{attribute 'GeneratedUsingTerminal: IODEVICETYPE_ETHERCATPROT'}
{attribute addProperty BoxType "IODEVICETYPE_ETHERCATPROT"}
{attribute addProperty Id "Beckhoff_EL1xxxBeckhoff_EL1xxx_3E37AACA6236Beckhoff_EL2xxxBeckhoff_EL2xxx_F4C539CA2992Beckhoff_EL3xxxBeckhoff_EL3xxx_05984D3D1813Beckhoff_EL3xxx_0030Beckhoff_EL3xxx_0030_EF742EC0265Beckhoff_EL4xxxBeckhoff_EL4xxx_BC7C1D702405Beckhoff_EL5xxxBeckhoff_EL5xxx_A510F2723086Beckhoff_EL6xxxBeckhoff_EL6xxx_5832F4A84115Beckhoff_EL7xxxBeckhoff_EL7xxx_96878FD52666Beckhoff_EL9xxxBeckhoff_EL9xxx_9771C92C1254Beckhoff_EL15xxBeckhoff_EL15xx_7FFDF3B3529Beckhoff_EL19xxBeckhoff_EL19xx_C9550BF750Beckhoff_EL25xxBeckhoff_EL25xx_A1E3F9182720Beckhoff_EL29xxBeckhoff_EL29xx_FCC67B4476Beckhoff_EL30xxBeckhoff_EL30xx_D5E79B105129Beckhoff_EL31xxBeckhoff_EL31xx_098DC56E3694Beckhoff_EL32xxBeckhoff_EL32xx_152143682581Beckhoff_EL33xxBeckhoff_EL33xx_7753F1402459Beckhoff_EL34xxBeckhoff_EL34xx_5C8507D711825Beckhoff_EL37xxBeckhoff_EL37xx_E7914E0E2253Beckhoff_EL47xxBeckhoff_EL47xx_F9F61196294Beckhoff_EL66xxBeckhoff_EL66xx_32F43B791034Beckhoff_EL67xxBeckhoff_EL67xx_9D033AAA966Beckhoff_EL68xxBeckhoff_EL68xx_6F2062753597Beckhoff_EL69xxBeckhoff_EL69xx_55DE5C9C198Beckhoff_EL72xxBeckhoff_EL72xx_566ED46D3383Beckhoff_EL73xxBeckhoff_EL73xx_3D4E24E01278Beckhoff_EL99xxBeckhoff_EL99xx_FA66A12D10SyncUnitsSyncUnits_9F8710E11242InputsInputs_25A0042B160OutputsOutputs_2397A10E106InfoDataInfoData_E68C61CD28"}
{attribute addProperty CRC "1261115388"}
{attribute addProperty Size "68444"}
TYPE EtherCAT_Master_ELxxxx_4B2B17FC :
STRUCT
	{attribute addProperty Name "Beckhoff_EL1xxx"}
	Beckhoff_EL1xxx : Beckhoff_EL1xxx_3E37AACA;
	{attribute addProperty Name "Beckhoff_EL2xxx"}
	Beckhoff_EL2xxx : Beckhoff_EL2xxx_F4C539CA;
	{attribute addProperty Name "Beckhoff_EL3xxx"}
	Beckhoff_EL3xxx : Beckhoff_EL3xxx_05984D3D;
	{attribute addProperty Name "Beckhoff_EL3xxx_0030"}
	Beckhoff_EL3xxx_0030 : Beckhoff_EL3xxx_0030_EF742EC0;
	{attribute addProperty Name "Beckhoff_EL4xxx"}
	Beckhoff_EL4xxx : Beckhoff_EL4xxx_BC7C1D70;
	{attribute addProperty Name "Beckhoff_EL5xxx"}
	Beckhoff_EL5xxx : Beckhoff_EL5xxx_A510F272;
	{attribute addProperty Name "Beckhoff_EL6xxx"}
	Beckhoff_EL6xxx : Beckhoff_EL6xxx_5832F4A8;
	{attribute addProperty Name "Beckhoff_EL7xxx"}
	Beckhoff_EL7xxx : Beckhoff_EL7xxx_96878FD5;
	{attribute addProperty Name "Beckhoff_EL9xxx"}
	Beckhoff_EL9xxx : Beckhoff_EL9xxx_9771C92C;
	{attribute addProperty Name "Beckhoff_EL15xx"}
	Beckhoff_EL15xx : Beckhoff_EL15xx_7FFDF3B3;
	{attribute addProperty Name "Beckhoff_EL19xx"}
	Beckhoff_EL19xx : Beckhoff_EL19xx_C9550BF7;
	{attribute addProperty Name "Beckhoff_EL25xx"}
	Beckhoff_EL25xx : Beckhoff_EL25xx_A1E3F918;
	{attribute addProperty Name "Beckhoff_EL29xx"}
	Beckhoff_EL29xx : Beckhoff_EL29xx_FCC67B44;
	{attribute addProperty Name "Beckhoff_EL30xx"}
	Beckhoff_EL30xx : Beckhoff_EL30xx_D5E79B10;
	{attribute addProperty Name "Beckhoff_EL31xx"}
	Beckhoff_EL31xx : Beckhoff_EL31xx_098DC56E;
	{attribute addProperty Name "Beckhoff_EL32xx"}
	Beckhoff_EL32xx : Beckhoff_EL32xx_15214368;
	{attribute addProperty Name "Beckhoff_EL33xx"}
	Beckhoff_EL33xx : Beckhoff_EL33xx_7753F140;
	{attribute addProperty Name "Beckhoff_EL34xx"}
	Beckhoff_EL34xx : Beckhoff_EL34xx_5C8507D7;
	{attribute addProperty Name "Beckhoff_EL37xx"}
	Beckhoff_EL37xx : Beckhoff_EL37xx_E7914E0E;
	{attribute addProperty Name "Beckhoff_EL47xx"}
	Beckhoff_EL47xx : Beckhoff_EL47xx_F9F61196;
	{attribute addProperty Name "Beckhoff_EL66xx"}
	Beckhoff_EL66xx : Beckhoff_EL66xx_32F43B79;
	{attribute addProperty Name "Beckhoff_EL67xx"}
	Beckhoff_EL67xx : Beckhoff_EL67xx_9D033AAA;
	{attribute addProperty Name "Beckhoff_EL68xx"}
	Beckhoff_EL68xx : Beckhoff_EL68xx_6F206275;
	{attribute addProperty Name "Beckhoff_EL69xx"}
	Beckhoff_EL69xx : Beckhoff_EL69xx_55DE5C9C;
	{attribute addProperty Name "Beckhoff_EL72xx"}
	Beckhoff_EL72xx : Beckhoff_EL72xx_566ED46D;
	{attribute addProperty Name "Beckhoff_EL73xx"}
	Beckhoff_EL73xx : Beckhoff_EL73xx_3D4E24E0;
	{attribute addProperty Name "Beckhoff_EL99xx"}
	Beckhoff_EL99xx : Beckhoff_EL99xx_FA66A12D;
	{attribute addProperty Name "SyncUnits"}
	SyncUnits : SyncUnits_9F8710E1;
	{attribute addProperty Name "Inputs"}
	Inputs : Inputs_25A0042B;
	{attribute addProperty Name "Outputs"}
	Outputs : Outputs_2397A10E;
	{attribute addProperty Name "InfoData"}
	InfoData : InfoData_E68C61CD;
END_STRUCT
END_TYPE

(* stored: Version 1.2.0.0, ProductVersion 3.1.4024.9
   DUT EtherCAT_Master_ELxxxx_4B2B17FC: Id {8d31f727-c815-4732-8aad-ca0ae42cb47d} *)
